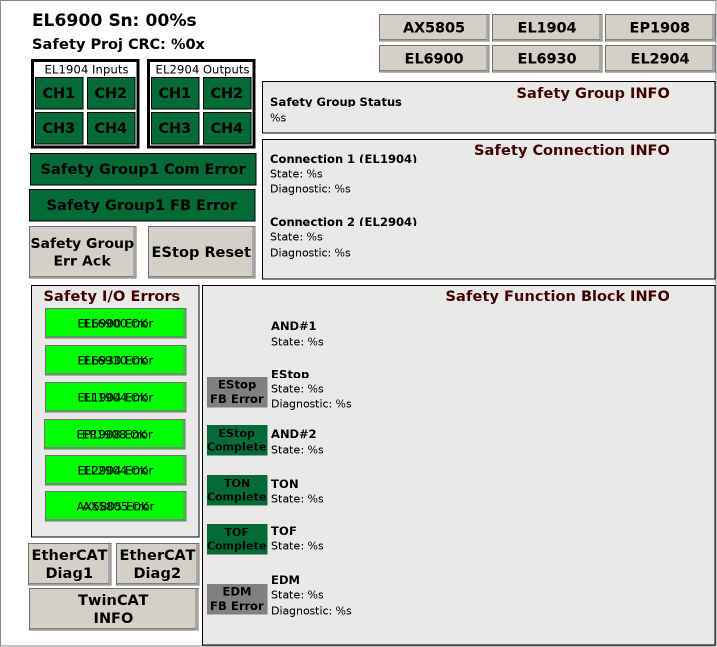
VISUALIZATION TwinSAFE  // 717x647
    RoundedRectangle (31,285 168x252)
    Rectangle (31,59 108x89)
    Rectangle (29,9 219x22), "EL6900 Sn: 00%s", text variable: g_udiHMI_SerialNumber
    Rectangle (29,33 232x22), "Safety Proj CRC: %0x", text variable: g_uiHMI_ProjectCRC
    Rectangle (35,77 48x32), "CH1", colour toggle: g_xHMI_EL1904Ch1
    Rectangle (87,77 48x32), "CH2", colour toggle: g_xHMI_EL1904Ch2
    Rectangle (35,112 48x32), "CH3", colour toggle: g_xHMI_EL1904Ch3
    Rectangle (87,112 48x32), "CH4", colour toggle: g_xHMI_EL1904Ch4
    Label (37,58 99x23), "EL1904 Inputs"
    Rectangle (147,59 108x89)
    Rectangle (151,77 48x32), "CH1", colour toggle: g_xHMI_EL2904Ch1
    Rectangle (203,77 48x32), "CH2", colour toggle: g_xHMI_EL2904Ch2
    Rectangle (151,112 48x32), "CH3", colour toggle: g_xHMI_EL2904Ch3
    Rectangle (203,112 48x32), "CH4", colour toggle: g_xHMI_EL2904Ch4
    Label (153,58 99x23), "EL2904 Outputs"
    Button (29,226 107x52), "Safety Group Err Ack"
        OnMouseDown: execute { g_xHMI_ErrAckPB := TRUE ; }
        OnMouseUp: execute { g_xHMI_ErrAckPB := FALSE ; }
    Button (148,226 107x52), "EStop Reset"
        OnMouseDown: execute { g_xHMI_EStopResetPB := TRUE ; }
        OnMouseUp: execute { g_xHMI_EStopResetPB := FALSE ; }
    Rectangle (30,153 226x32), "Safety Group1 Com Error", colour toggle: g_xHMI_SafetyGroup1_COMerrorLT
    Rectangle (29,189 226x32), "Safety Group1 FB Error", colour toggle: g_xHMI_SafetyGroup1_FBerrorLT
    Label (50,283 133x26), "Safety I/O Errors"
    Button (28,543 83x42), "EtherCAT Diag1"
        OnMouseClick: change screen: EtherCAT_Diag1
    Button (116,543 83x42), "EtherCAT Diag2"
        OnMouseClick: change screen: EtherCAT_Diag2
    Button (29,588 169x42), "TwinCAT INFO"
        OnMouseClick: change screen: TwinCAT_INFO
    RoundedRectangle (262,81 453x52)
    Label (449,80 224x26), "Safety Group INFO"
    Label (267,89 135x26), "Safety Group Status"
    RoundedRectangle (262,139 453x140)
    Label (449,137 224x26), "Safety Connection INFO"
    Label (267,146 203x26), "Connection 1 (EL1904)"
    Label (267,209 203x26), "Connection 2 (EL2904)"
    RoundedRectangle (202,285 513x360)
    Label (449,283 224x26), "Safety Function Block INFO"
    Label (268,313 50x26), "AND#1"
    Label (268,362 51x25), "EStop"
    Button (379,14 110x27), "AX5805"
        OnMouseClick: change screen: AX5805_Specific_Diagnostics
    Button (379,45 110x27), "EL6900"
        OnMouseClick: change screen: EL6900_Specific_Diagnostics
    Button (492,14 110x27), "EL1904"
        OnMouseClick: change screen: EL1904_Specific_Diagnostics
    Button (492,45 110x27), "EL6930"
        OnMouseClick: change screen: EL6930_Specific_Diagnostics
    Button (605,14 110x27), "EP1908"
        OnMouseClick: change screen: EP1908_Specific_Diagnostics
    Button (605,45 110x27), "EL2904"
        OnMouseClick: change screen: EL2904_Specific_Diagnostics
    Rectangle (267,107 321x22), "%s", text variable: g_sHMI_StatusGroup1
    Rectangle (267,163 321x22), "State: %s", text variable: g_sHMI_StateConn1
    Rectangle (267,178 386x22), "Diagnostic: %s", text variable: g_sHMI_DiagConn1
    Rectangle (267,226 321x22), "State: %s", text variable: g_sHMI_StateConn2
    Rectangle (267,242 389x22), "Diagnostic: %s", text variable: g_sHMI_DiagConn2
    Rectangle (268,331 439x22), "State: %s", text variable: g_sHMI_StatusAND1
    Rectangle (268,378 439x22), "State: %s", text variable: g_sHMI_StatusEStop1
    Rectangle (268,393 439x22), "Diagnostic: %s", text variable: g_sHMI_DiagEStop1
    Rectangle (268,439 439x22), "State: %s", text variable: g_sHMI_StatusAND2
    Label (268,421 54x26), "AND#2"
    Rectangle (268,488 439x22), "State: %s", text variable: g_sHMI_StatusTON
    Label (268,471 36x26), "TON"
    Rectangle (268,535 439x22), "State: %s", text variable: g_sHMI_StatusTOF
    Label (268,518 33x26), "TOF"
    Label (268,571 34x18), "EDM"
    Rectangle (268,584 439x22), "State: %s", text variable: g_sHMI_StatusEDM
    Rectangle (268,600 439x22), "Diagnostic: %s", text variable: g_sHMI_DiagEDM
    Rectangle (207,377 60x30), "EStop FB Error", colour toggle: g_xHMI_EStop_errorLT
    Rectangle (207,425 60x30), "EStop Complete", colour toggle: g_xHMI_EStop_CompleteLT
    Rectangle (207,475 60x30), "TON Complete", colour toggle: g_xHMI_EStop_ON_Delay_CompleteLT
    Rectangle (207,524 60x30), "TOF Complete", colour toggle: g_xHMI_EStop_OFF_Delay_CompleteLT
    Rectangle (207,584 60x30), "EDM FB Error", colour toggle: g_xHMI_EDMerrorLT
    Group (45,308 141x30)
        Button (0,0 141x30), colour toggle: g_xHMI_EL6900_General_Error
            OnMouseClick: change screen: AX5805_Specific_Diagnostics
            OnMouseUp: execute { g_xHMI_ErrAckPB := FALSE ; }
        Label (10,3 121x25), "EL6900 Error", invisible if: NOT g_xHMI_EL6900_General_Error
        Label (10,3 121x25), "EL6900 OK", invisible if: g_xHMI_EL6900_General_Error
    Group (45,345 141x30)
        Button (0,0 141x30), colour toggle: g_xHMI_EL6930_General_Error
            OnMouseClick: change screen: AX5805_Specific_Diagnostics
            OnMouseUp: execute { g_xHMI_ErrAckPB := FALSE ; }
        Label (10,3 121x25), "EL6930 Error", invisible if: NOT g_xHMI_EL6930_General_Error
        Label (10,3 121x25), "EL6930 OK", invisible if: g_xHMI_EL6930_General_Error
    Group (45,382 141x30)
        Button (0,0 141x30), colour toggle: g_xHMI_EL1904_General_Error
            OnMouseClick: change screen: AX5805_Specific_Diagnostics
            OnMouseUp: execute { g_xHMI_ErrAckPB := FALSE ; }
        Label (10,3 121x25), "EL1904 Error", invisible if: NOT g_xHMI_EL1904_General_Error
        Label (10,3 121x25), "EL1904 OK", invisible if: g_xHMI_EL1904_General_Error
    Group (44,419 141x30)
        Button (0,0 141x30), colour toggle: g_xHMI_EP1908_General_Error
            OnMouseClick: change screen: AX5805_Specific_Diagnostics
            OnMouseUp: execute { g_xHMI_ErrAckPB := FALSE ; }
        Label (10,3 121x25), "EP1908 Error", invisible if: NOT g_xHMI_EP1908_General_Error
        Label (10,3 121x25), "EP1908 OK", invisible if: g_xHMI_EP1908_General_Error
    Group (45,455 141x30)
        Button (0,0 141x30), colour toggle: g_xHMI_EL2904_General_Error
            OnMouseClick: change screen: AX5805_Specific_Diagnostics
            OnMouseUp: execute { g_xHMI_ErrAckPB := FALSE ; }
        Label (10,3 121x25), "EL2904 Error", invisible if: NOT g_xHMI_EL2904_General_Error
        Label (10,3 121x25), "EL2904 OK", invisible if: g_xHMI_EL2904_General_Error
    Group (45,491 141x30)
        Button (0,0 141x30), colour toggle: g_xHMI_AX5805_General_Error
            OnMouseClick: change screen: AX5805_Specific_Diagnostics
            OnMouseUp: execute { g_xHMI_ErrAckPB := FALSE ; }
        Label (10,3 121x25), "AX5805 Error", invisible if: NOT g_xHMI_AX5805_General_Error
        Label (10,3 121x25), "AX5805 OK", invisible if: g_xHMI_AX5805_General_Error
END_VISUALIZATION

(* stored: Version 1.1.0.1, ProductVersion 3.1.0.18
   Visu TwinSAFE: Id {a4d5bb29-e369-453d-bc62-6d8ba81dbeb6} *)
